FUNCTION_BLOCK FB_System_MVWW_245
VAR_INPUT

	Freigabe_auto			: BOOL;
	Freigabe_Deakt_auto		: BOOL;
	Betrieb_Anford_auto		: BOOL;

	Regelung_Modus_auto		: SINT;
	Regelung_Sollw_auto		: REAL;
END_VAR
VAR_OUTPUT

	{attribute 'OPC.UA.DA' := '1'}Parameter		: ST_System_MVWW_Parameter;  
	{attribute 'OPC.UA.DA' := '1'}Zustand			: ST_System_MVWW_Zustand;
	{attribute 'OPC.UA.DA' := '1'}Stellwert		: ST_System_MVWW_Stellwert;	 
	{attribute 'OPC.UA.DA' := '1'}Steuerung		: ST_System_MVWW_Steuerung;	 
END_VAR
VAR
	Pumpe_245		:FB_PU;
	Stellventil_245	:FB_SV;

	Ablaufsteuerung	: FB_System_MVWW_Ablaufsteuerung;
	Logik			: FB_System_MVWW_Logik;
	Zustandscheck	: FB_System_MVWW_Zustandscheck;
	Stellwertscheck	: FB_System_MVWW_Stellwertscheck;
	Sollwertscheck	: FB_System_MVWW_Sollwertscheck;
	DC_Schaltschrank: FB_DCSS;
	EMAG_VLC100Y	: FB_MV_EMAG_VLC100Y;
	Chiller			: FB_KKKW;
END_VAR
VAR // added by the converter: edge detectors and wires of the graphical bodies
    _w1, _w2 : ANY;
END_VAR

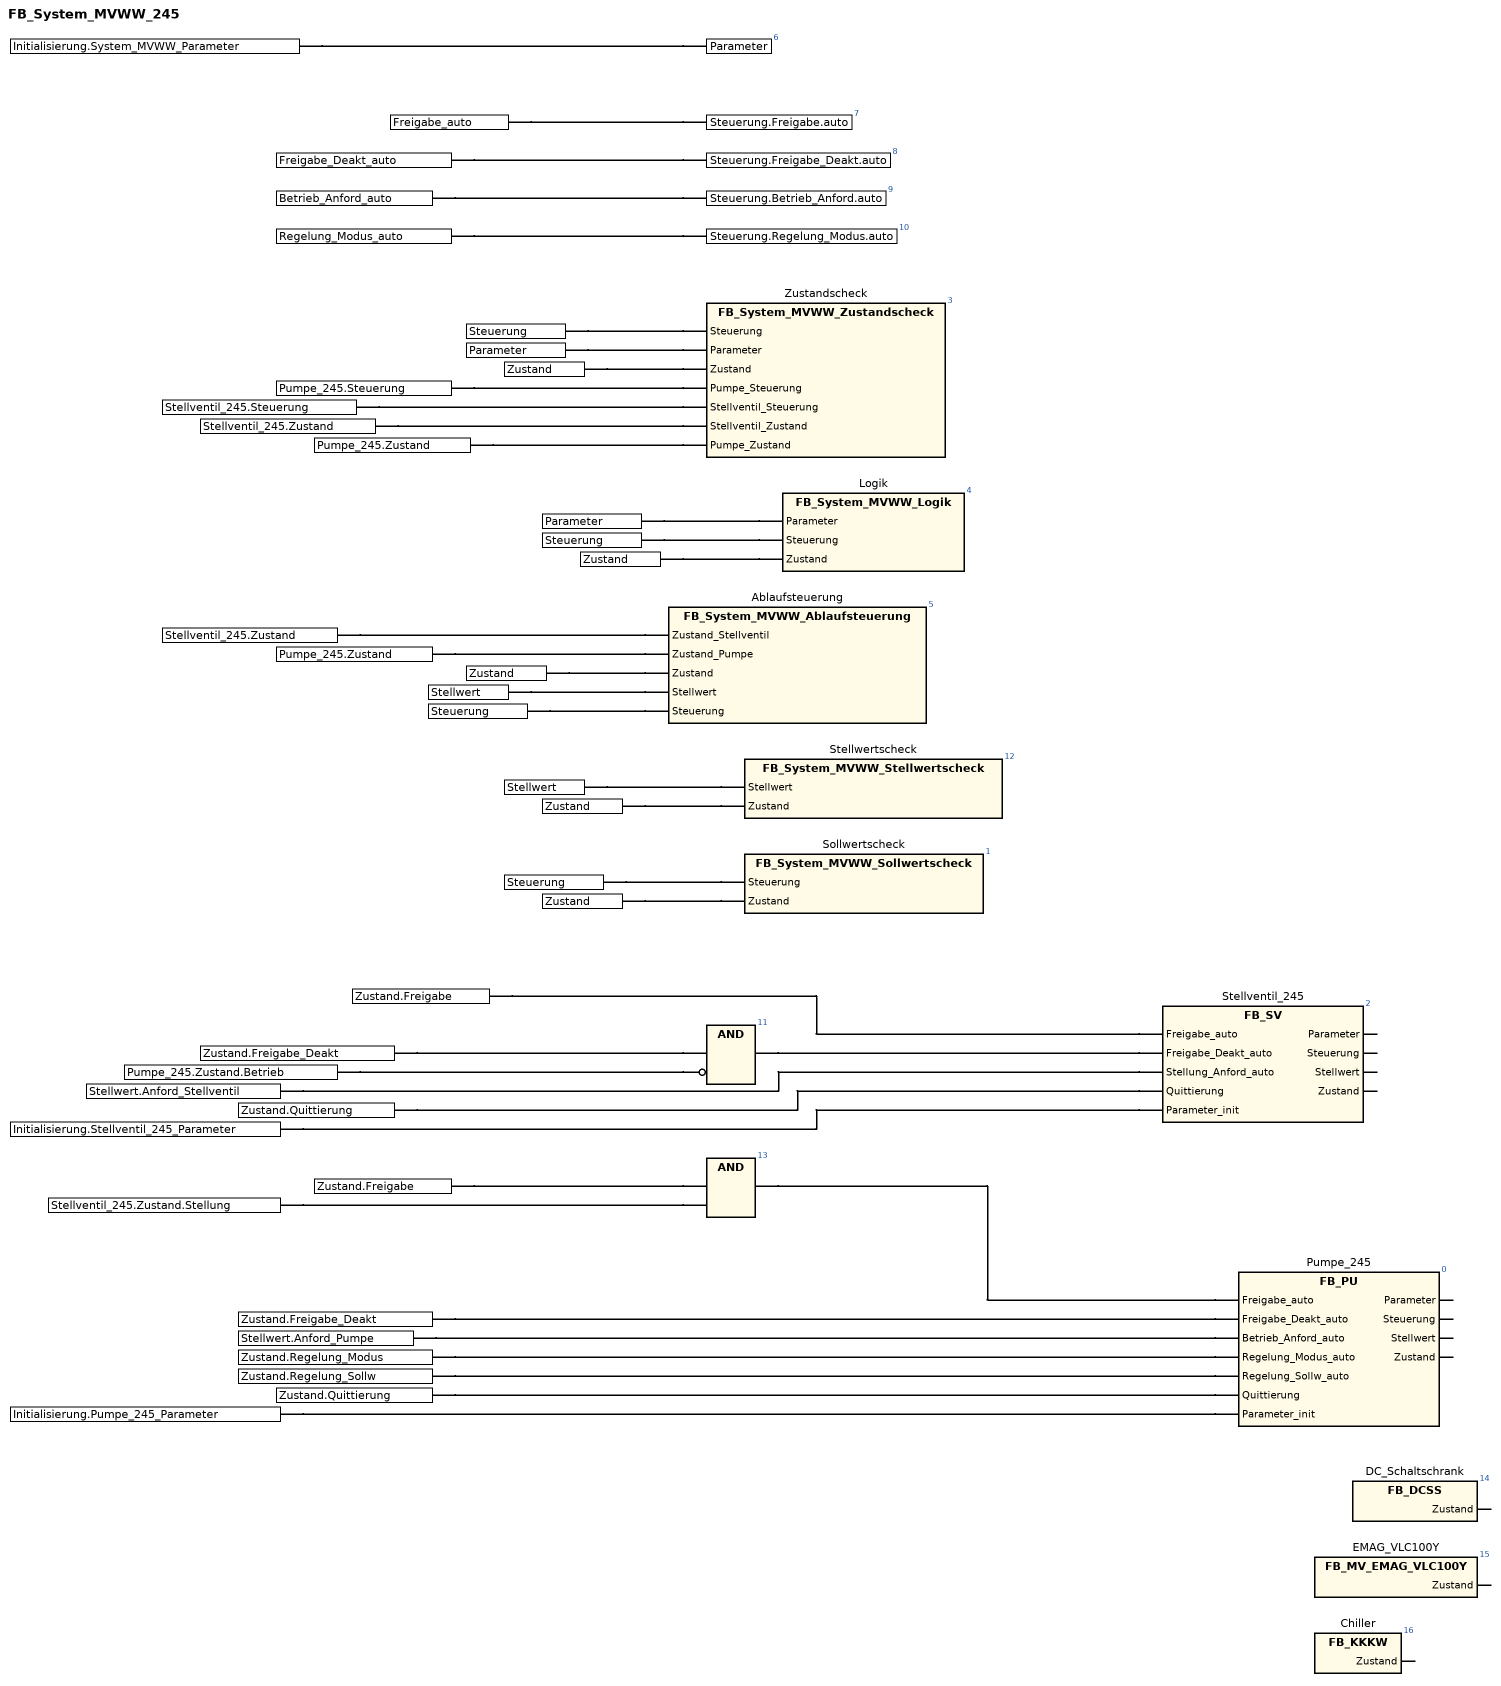
Pumpe_245(
    Freigabe_auto := _w1,
    Freigabe_Deakt_auto := Zustand.Freigabe_Deakt,
    Betrieb_Anford_auto := Stellwert.Anford_Pumpe,
    Regelung_Modus_auto := Zustand.Regelung_Modus,
    Regelung_Sollw_auto := Zustand.Regelung_Sollw,
    Quittierung := Zustand.Quittierung,
    Parameter_init := Initialisierung.Pumpe_245_Parameter); // FB_PU
Sollwertscheck(Steuerung := Steuerung, Zustand := Zustand); // FB_System_MVWW_Sollwertscheck
Stellventil_245(
    Freigabe_auto := Zustand.Freigabe,
    Freigabe_Deakt_auto := _w2,
    Stellung_Anford_auto := Stellwert.Anford_Stellventil,
    Quittierung := Zustand.Quittierung,
    Parameter_init := Initialisierung.Stellventil_245_Parameter); // FB_SV
Zustandscheck(
    Steuerung := Steuerung,
    Parameter := Parameter,
    Zustand := Zustand,
    Pumpe_Steuerung := Pumpe_245.Steuerung,
    Stellventil_Steuerung := Stellventil_245.Steuerung,
    Stellventil_Zustand := Stellventil_245.Zustand,
    Pumpe_Zustand := Pumpe_245.Zustand); // FB_System_MVWW_Zustandscheck
Logik(Parameter := Parameter, Steuerung := Steuerung, Zustand := Zustand); // FB_System_MVWW_Logik
Ablaufsteuerung(
    Zustand_Stellventil := Stellventil_245.Zustand,
    Zustand_Pumpe := Pumpe_245.Zustand,
    Zustand := Zustand,
    Stellwert := Stellwert,
    Steuerung := Steuerung); // FB_System_MVWW_Ablaufsteuerung
Parameter := Initialisierung.System_MVWW_Parameter;
Steuerung.Freigabe.auto := Freigabe_auto;
Steuerung.Freigabe_Deakt.auto := Freigabe_Deakt_auto;
Steuerung.Betrieb_Anford.auto := Betrieb_Anford_auto;
Steuerung.Regelung_Modus.auto := Regelung_Modus_auto;
_w2 := Zustand.Freigabe_Deakt AND NOT Pumpe_245.Zustand.Betrieb;
Stellwertscheck(Stellwert := Stellwert, Zustand := Zustand); // FB_System_MVWW_Stellwertscheck
_w1 := Zustand.Freigabe AND Stellventil_245.Zustand.Stellung;
DC_Schaltschrank(); // FB_DCSS
EMAG_VLC100Y(); // FB_MV_EMAG_VLC100Y
Chiller(); // FB_KKKW

END_FUNCTION_BLOCK

(* stored: Version 1.1.0.1, ProductVersion 3.1.4024.9
   POU FB_System_MVWW_245: Id {f7c3b010-c852-47b8-a7cb-d8d52c1491f8}, SpecialFunc None *)
